TEXTLIST Noms_Modes
  1 = 'DOUCHE BONDE OUVERTE ET TEMPO' | En: 'SHOWER WITH DRAIN AND DELAY'
  2 = 'DOUCHE BONDE FERMEE ET TEMPO' | En: 'SHOWER WITHOUT DRAIN AND DELAY'
  3 = 'DOUCHETTE' | En: 'CLEANING'
  4 = 'LAVABO BONDE OUVERTE ET TEMPO' | En: 'SINK WITH DRAIN AND DELAY'
  5 = 'LAVABO BONDE FERMEE ET TEMPO' | En: 'SINK WITHOUT DRAIN AND DELAY'
  6 = 'PRISE ELECTRIQUE' | En: 'PLUG ACTIVATE'
  7 = 'VIDANGE(S)' | En: 'OPENED DRAIN'
  8 = 'NEUTRE' | En: 'NEUTRAL'
  9 = 'CHASSE D EAU GRAND VOLUME' | En: 'LARGE VOLUME TOILET FLUSH'
  10 = 'DEPOLLUTION' | En: 'DECONTAMINATION'
  11 = 'NEUTRE AVEC BAS DEBIT' | En: 'NEUTRAL WITH LOW FLOW'
  12 = 'DOUCHE BONDE OUVERTE ET VOLUME' | En: 'SHOWER WITH DRAIN AND VOLUME'
  13 = 'DOUCHE BONDE FERMEE ET VOLUME' | En: 'SHOWER WITHOUT DRAIN AND VOLUME'
  14 = 'LAVABO BONDE OUVERTE ET VOLUME' | En: 'SINK WITH DRAIN AND VOLUME'
  15 = 'LAVABO BONDE FERMEE ET VOLUME' | En: 'SINK WITHOUT DRAIN AND VOLUME'
  16 = 'DOUCHE BONDE OUVERTE ET BOUTON' | En: 'SHOWER WITH DRAIN AND BUTTON'
  17 = 'LAVABO BONDE OUVERTE ET BOUTON' | En: 'SINK WITH DRAIN AND BUTTON'
  18 = 'LAVAGE CHAUD' | En: 'HOT CLEANING'
  19 = 'LAVAGE FROID' | En: 'COLD CLEANING'
  20 = 'MODE PARAMETRABLE' | En: 'PARAMETER MODE'
  21 = 'ALERTE PREPARATEUR' | En: 'PREPARATOR ALERT'
  22 = 'ALERTE EVALUATEUR' | En: 'EVALUATOR ALERT'
  23 = 'EVALUATION' | En: 'EVALUATION'
  24 = 'EVALUATION AVEC AIR' | En: 'EVALUATION WITH AIR FLOW'
  25 = 'MISE EN CONDITION' | En: 'CONDITIONING BOOTH'
  26 = 'CHASSE D EAU PETIT VOLUME' | En: 'SMALL VOLUME TOILET FLUSH'
  27 = 'LAVAGE NEP' | En: 'CLEANING'
  28 = 'CABINE EN CONDITION' | En: 'BOOTH IN CONDITION'
  29 = 'LIBRE' | En: 'EMPTY'
  30 = 'MODE TEXTE' | En: 'TEXT MODE'
  0 = ''
   = ''
END_TEXTLIST

(* stored: Version 1.1.0.1, ProductVersion 3.1.4024.15
   TextList Noms_Modes: Id {e8e0f21e-9ec3-4820-bf71-bc64e873a4a1} *)
